KUKA KRL program: TEST_ToolMeasure.src, TEST_ToolMeasure.dat

--- TEST_ToolMeasure.src ---
&ACCESS RVO
&REL 58
&PARAM DISKPATH = KRC:\R1\Program\Test\ToolMagazine
DEF TEST_ToolMeasure( )
   ;FOLD DECL
      DECL POS xAboveSensor,xMeasureStart,xMeasureEnd
      DECL FRAME fStartOffset,fEndOffset
   ;ENDFOLD
   ;FOLD INI
      xAboveSensor = fAboveSensor:xSensor

      fStartOffset = $NULLFRAME
      fStartOffset.Z = rToolLengthMax + rMeasureOffset
      xMeasureStart = fStartOffset:xSensor

      fEndOffset = $NULLFRAME
      fEndOffset.Z = rToolLengthMin - rMeasureOffset
      xMeasureEnd = fEndOffset:xSensor

      rToolLength = -1

      INTERRUPT DECL iSafetyStop WHEN NOT inToolLengthSafeSwitch DO SafetyStop()
      INTERRUPT DECL iMeasureStop WHEN NOT inToolLengthSwitch DO MeasureStop()
   ;ENDFOLD

   IF NOT (inToolLengthSafeSwitch AND inToolLengthSwitch) THEN
      HALT ;Nieprawidłowy stan czujnika
   ENDIF
   INTERRUPT ON iSafetyStop

   SetBaseTool(#ToolMagazine,#Spindle1)
   SetVel(#SpindleIdle)
   LIN xAboveSensor C_DIS
   LIN xMeasureStart

   WAIT SEC 0
   Measure(xMeasureEnd)

   SetVel(#SpindleIdle)
   LIN_REL fToolMeasured
   ;Sprawdzać czy czujnik wrocił do stanu pierwotnego?
   LIN xMeasureStart C_DIS
   LIN xAboveSensor

   WAIT SEC 1
   INTERRUPT OFF iSafetyStop
   ShowLength()
   ;TODO - Aktualizacja długosci mierzonego narzędzia
   WAIT SEC 1
   HALT

END

DEF Measure(xMeasureEnd:IN)
   DECL POS xMeasureEnd

   IF NOT inToolLengthSwitch THEN
      HALT ;Niepoprawny stan czujnika
   ENDIF

   SetVel(#ToolMeasure)
   INTERRUPT ON iMeasureStop
   LIN xMeasureEnd
   WAIT SEC 0
   HALT  ;Ruch pomiaru nie został przerwany
END

DEF SafetyStop()
   ;Osiągnięcie maksymalnej pozycji czujnika długoSci narzędzia
   BRAKE F
   WAIT SEC 3
   HALT
END

DEF MeasureStop()
   ;Dotknięcia powierzchni czujnika długoSci narzędzia
   DECL FRAME fTool

   xSpindle = $POS_INT
   BRAKE
   INTERRUPT OFF iMeasureStop
   fTool = INV_POS(xSensor):xSpindle
   rToolLength = fTool.z

   IF (rToolLength<rToolLengthMin) OR (rToolLength>rToolLengthMax) THEN
      HALT  ;DługoSć narzędzia poza zakresem
   ENDIF

   RESUME
END

DEF ShowLength()
   ;WyScietlenie zmierzonej długoSci narzędzia
   DECL INT nAnswer,iOffset
   DECL CHAR sToolLength[20]
   DECL STATE_T STATE
   DECL REAL rWartosc

   iOffset = 0

   SWRITE(sToolLength[],STATE,iOffset,"%.2f",rToolLength)
   MsgDialog(nAnswer,"Zmierzona dlugosc narzedzia %1 mm","ToolMeasure",sToolLength[],"OK")

END

--- TEST_ToolMeasure.dat ---
&ACCESS RVO
&REL 58
&PARAM DISKPATH = KRC:\R1\Program\Test\ToolMagazine
DEFDAT  TEST_ToolMeasure

DECL CONST INT iSafetyStop=11
DECL CONST INT iMeasureStop=12

DECL POS xSpindle
DECL REAL rToolLength=-1.00000

DECL CONST REAL rToolLengthMin=120.000
DECL CONST REAL rToolLengthMax=230.000
DECL CONST REAL rMeasureOffset=10.0000

DECL CONST POS xSensor={X 725.700,Y -70.5000,Z 63.6000,A 0.0,B 0.0,C 0.0}
DECL CONST FRAME fAboveSensor={X 0.0,Y 0.0,Z 300.000,A 0.0,B 0.0,C 0.0}
DECL CONST FRAME fMeasureOffset={X 0.0,Y 0.0,Z 10.0000,A 0.0,B 0.0,C 0.0}

DECL CONST FRAME fMeasureStart={X 0.0,Y 0.0,Z 250.000,A 0.0,B 0.0,C 0.0}
DECL CONST FRAME fMeasureEnd={X 0.0,Y 0.0,Z 100.000,A 0.0,B 0.0,C 0.0}

DECL CONST FRAME fToolMeasured={X 0.0,Y 0.0,Z 15.0000,A 0.0,B 0.0,C 0.0}

ENDDAT
